SYSTEM TEST_TAGS (* Test TAGIN and TAGOUT types *)
  (* Standard: 61499-1 *)
  (* Version 0.0, 2007-01-13, JHC, Holobloc Inc *)
  DEVICE PUBLISHER : FRAME_DEVICE(GRID := [3,1], BOUNDS := [100,100,150,200])
    RESOURCE MGR : RMT_RES
    END_RESOURCE
    RESOURCE TEST0 : PANEL_RESOURCE
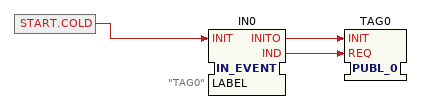
      FBS
        IN0 : IN_EVENT(LABEL := "TAG0");
        TAG0 : PUBL_0; (* Pure Event *)
      END_FBS
      EVENT_CONNECTIONS
        START.COLD TO IN0.INIT;
        IN0.INITO TO TAG0.INIT;
        IN0.IND TO TAG0.REQ;
      END_CONNECTIONS
    END_RESOURCE
    RESOURCE TEST1 : PANEL_RESOURCE
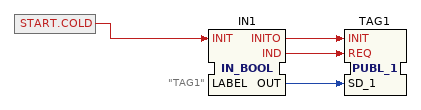
      FBS
        IN1 : IN_BOOL(LABEL := "TAG1");
        TAG1 : PUBL_1;
      END_FBS
      EVENT_CONNECTIONS
        START.COLD TO IN1.INIT;
        IN1.INITO TO TAG1.INIT;
        IN1.IND TO TAG1.REQ;
      END_CONNECTIONS
      DATA_CONNECTIONS
        IN1.OUT TO TAG1.SD_1;
      END_CONNECTIONS
    END_RESOURCE
    RESOURCE TEST2 : PANEL_RESOURCE
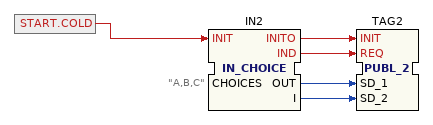
      FBS
        IN2 : IN_CHOICE(CHOICES := "A,B,C");
        TAG2 : PUBL_2; (* Tag Group with 2 values *)
      END_FBS
      EVENT_CONNECTIONS
        START.COLD TO IN2.INIT;
        IN2.INITO TO TAG2.INIT;
        IN2.IND TO TAG2.REQ;
      END_CONNECTIONS
      DATA_CONNECTIONS
        IN2.OUT TO TAG2.SD_1;
        IN2.I TO TAG2.SD_2;
      END_CONNECTIONS
    END_RESOURCE
    RESOURCE TAGS : EMB_RES
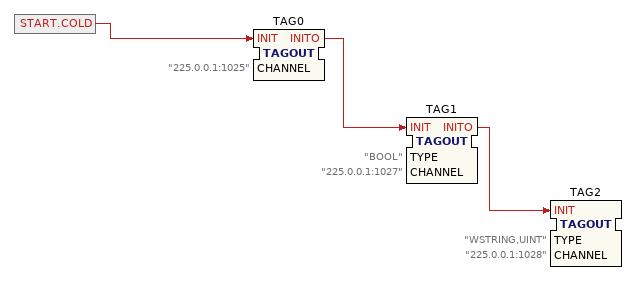
      FBS
        TAG0 : TAGOUT(CHANNEL := "225.0.0.1:1025");
        TAG1 : TAGOUT(TYPE := "BOOL", CHANNEL := "225.0.0.1:1027");
        TAG2 : TAGOUT(TYPE := "WSTRING,UINT", CHANNEL := "225.0.0.1:1028"); (* Tag Group with 2 values *)
      END_FBS
      EVENT_CONNECTIONS
        START.COLD TO TAG0.INIT;
        TAG0.INITO TO TAG1.INIT;
        TAG1.INITO TO TAG2.INIT;
      END_CONNECTIONS
    END_RESOURCE
  END_DEVICE
  DEVICE SUBSCRIBER : RMT_FRAME(BOUNDS := [250,100,150,200], GRID := [3,1])
    RESOURCE MGR : RMT_RES
    END_RESOURCE
    RESOURCE TEST0 : PANEL_RESOURCE
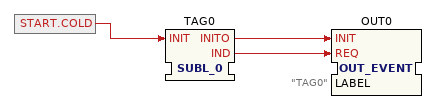
      FBS
        TAG0 : SUBL_0;
        OUT0 : OUT_EVENT(LABEL := "TAG0");
      END_FBS
      EVENT_CONNECTIONS
        START.COLD TO TAG0.INIT;
        TAG0.INITO TO OUT0.INIT;
        TAG0.IND TO OUT0.REQ;
      END_CONNECTIONS
    END_RESOURCE
    RESOURCE TEST1 : PANEL_RESOURCE
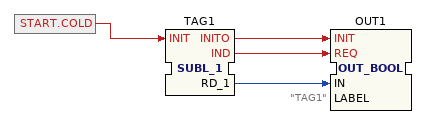
      FBS
        TAG1 : SUBL_1;
        OUT1 : OUT_BOOL(LABEL := "TAG1");
      END_FBS
      EVENT_CONNECTIONS
        START.COLD TO TAG1.INIT;
        TAG1.INITO TO OUT1.INIT;
        TAG1.IND TO OUT1.REQ;
      END_CONNECTIONS
      DATA_CONNECTIONS
        TAG1.RD_1 TO OUT1.IN;
      END_CONNECTIONS
    END_RESOURCE
    RESOURCE TEST2 : PANEL_RESOURCE
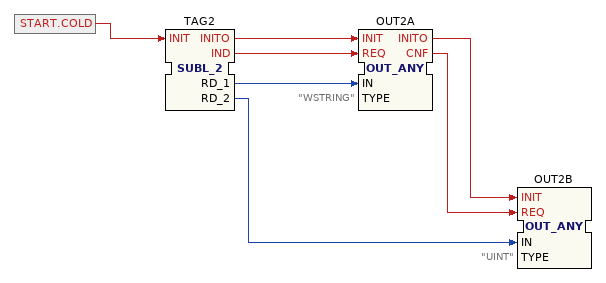
      FBS
        TAG2 : SUBL_2;
        OUT2A : OUT_ANY(TYPE := "WSTRING");
        OUT2B : OUT_ANY(TYPE := "UINT");
      END_FBS
      EVENT_CONNECTIONS
        START.COLD TO TAG2.INIT;
        TAG2.INITO TO OUT2A.INIT;
        OUT2A.INITO TO OUT2B.INIT;
        TAG2.IND TO OUT2A.REQ;
        OUT2A.CNF TO OUT2B.REQ;
      END_CONNECTIONS
      DATA_CONNECTIONS
        TAG2.RD_1 TO OUT2A.IN;
        TAG2.RD_2 TO OUT2B.IN;
      END_CONNECTIONS
    END_RESOURCE
    RESOURCE TAGS : EMB_RES
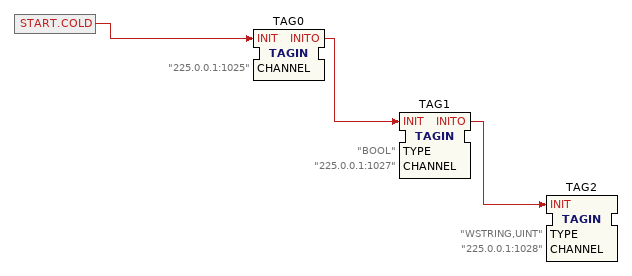
      FBS
        TAG0 : TAGIN(CHANNEL := "225.0.0.1:1025");
        TAG1 : TAGIN(TYPE := "BOOL", CHANNEL := "225.0.0.1:1027");
        TAG2 : TAGIN(TYPE := "WSTRING,UINT", CHANNEL := "225.0.0.1:1028"); (* Tag Group with 2 values *)
      END_FBS
      EVENT_CONNECTIONS
        START.COLD TO TAG0.INIT;
        TAG0.INITO TO TAG1.INIT;
        TAG1.INITO TO TAG2.INIT;
      END_CONNECTIONS
    END_RESOURCE
  END_DEVICE
END_SYSTEM
